PROGRAM MaintenanceTask
VAR
	CycleCounter: INT := 0;;
	MaintenanceNeeded: BOOL;
	Message: STRING(INT#16);
	Tclean: Ton;
	
	ResetCounter: BOOL;
	CoffeeReadyOld: BOOL := FALSE;
	
END_VAR

// every cooffee made the counter increase
IF (GVL.CoffeeReady = TRUE) AND (CoffeeReadyOld = FALSE) THEN
    CycleCounter := CycleCounter + 1;
END_IF;

CoffeeReadyOld := GVL.CoffeeReady;

// if the machine has done 5 coffee, the cleaning part is needed
IF CycleCounter >= 5 THEN
    MaintenanceNeeded := TRUE;
    Message := 'Maintenance required!';
	GVL.CLEANING := TRUE;

    Tclean(IN := TRUE, PT := T#4S);

    IF Tclean.Q THEN
        Tclean(IN := FALSE);
        ResetCounter := TRUE;
    END_IF;
//maintenance finished and numbur of coffe made
ELSE
    MaintenanceNeeded := FALSE;
    Message := CONCAT('Coffees made: ', INT_TO_STRING(CycleCounter));
	GVL.CLEANING := FALSE;
END_IF;

//after cleaning, counter must be resetted
IF ResetCounter = TRUE THEN  
    CycleCounter := 0;
    MaintenanceNeeded := FALSE;
    Message := 'Maintenance done';
    ResetCounter := FALSE; 
END_IF;

END_PROGRAM

(* stored: Version 1.1.0.1, ProductVersion 3.1.4024.15
   POU MaintenanceTask: Id {f2ccf1d7-5961-4f5a-bde9-3b71431e1174}, SpecialFunc None *)
